TYPE E_HomeX :
(
	Init := 0,
    Power_On :=1,
    Check_Homed :=2,
    Home_X1 :=3,
    X1_Homed :=4,
    Home_X2 :=5,
    X2_Homed :=6,
    Gear_In :=7,
    End_Sequence :=8
    
);
END_TYPE

(* stored: Version 1.1.0.1, ProductVersion 3.1.4024.3
   DUT E_HomeX: Id {7737f691-b37c-43b8-aec3-3723fe7e4366} *)
